CASE state OF
    BAG_DELIVERY_STATES.Idle :                     
													IF _mode = DEVICE_MODES.Manual THEN 
														state := BAG_DELIVERY_STATES.Manual;
													ELSIF NOT iBagNotPresent OR Globals.enableDryCycle THEN
														state := BAG_DELIVERY_STATES.Ready;
													ELSIF iBagNotPresent AND (_amFeedToEye OR _amReverseBag) THEN
														state := BAG_DELIVERY_STATES.FeedToEye;
														_amFeedToEye := FALSE;
													END_IF
													IF jogForwardONS.OSR THEN
														bagFeedMasterMotor.MoveDistance(distance := 30, 
                                                                                    acceleration := accelSetpoint, 
                                                                                    deceleration := decelSetpoint, 
                                                                                    velocity := REAL_TO_INT((1 * Globals.VELOCITY_IPS_MULTIPLIER_20_DEGREE_BAG_DELIVERY)));
														bagFeedRearMotor.MoveDistance(distance := 30, 
                                                                                    acceleration := accelSetpoint, 
                                                                                    deceleration := decelSetpoint, 
                                                                                    velocity := REAL_TO_INT((1 * Globals.VELOCITY_IPS_MULTIPLIER_20_DEGREE_BAG_DELIVERY)));
													ELSIF jogReverseONS.OSR THEN
														bagFeedMasterMotor.MoveDistance(distance := -30, 
                                                                                    acceleration := accelSetpoint, 
                                                                                    deceleration := decelSetpoint, 
                                                                                    velocity := REAL_TO_INT((1 * Globals.VELOCITY_IPS_MULTIPLIER_20_DEGREE_BAG_DELIVERY)));
														bagFeedRearMotor.MoveDistance(distance := -30, 
                                                                                    acceleration := accelSetpoint, 
                                                                                    deceleration := decelSetpoint, 
                                                                                    velocity := REAL_TO_INT((1 * Globals.VELOCITY_IPS_MULTIPLIER_20_DEGREE_BAG_DELIVERY)));
													ELSIF jogForwardONS.OSF OR jogReverseONS.OSF THEN
														bagFeedMasterMotor.Stop();
														bagFeedRearMotor.Stop();
													END_IF
    
	BAG_DELIVERY_STATES.FeedToEye :					//Feed to photoeye if not present
													bagFeedMasterMotor.MoveDistance(distance := feedToPhotoeyeSetpoint, 
                                                                                    acceleration := accelSetpoint, 
                                                                                    deceleration := decelSetpoint, 
                                                                                    velocity := REAL_TO_INT((feedToPhotoeyeSetpoint * Globals.VELOCITY_IPS_MULTIPLIER_20_DEGREE_BAG_DELIVERY)));
													bagFeedRearMotor.MoveDistance(distance := feedToPhotoeyeSetpoint, 
                                                                                    acceleration := accelSetpoint, 
                                                                                    deceleration := decelSetpoint, 
                                                                                    velocity := REAL_TO_INT((feedToPhotoeyeSetpoint * Globals.VELOCITY_IPS_MULTIPLIER_20_DEGREE_BAG_DELIVERY)));
													state := BAG_DELIVERY_STATES.FeedingToEye;
													
	BAG_DELIVERY_STATES.FeedingToEye :				// Stop once photoeye seen
													delay.PT := T#3S;
													delay.IN := TRUE;
													IF NOT iBagNotPresent THEN
														bagFeedMasterMotor.Stop();
														bagFeedRearMotor.Stop();
														state := BAG_DELIVERY_STATES.Idle;
														delay.IN := FALSE;
													END_IF
													IF delay.Q THEN
														state := BAG_DELIVERY_STATES.Fault;
														noBagOverEye.Trigger();
														delay.IN := FALSE;
													END_IF
	
    BAG_DELIVERY_STATES.Reverse :                    // Reverse to break perf
                                                    bagFeedMasterMotor.MoveDistance(distance := reverseDistanceSetpoint, 
                                                                                    acceleration := TO_INT((ABS(reverseDistanceSetpoint) * Globals.STEPS_PER_INCH_20_DEGREE_BAG_DELIVERY) *  accelPercent),
                                                                                    deceleration := TO_INT((ABS(reverseDistanceSetpoint) * Globals.STEPS_PER_INCH_20_DEGREE_BAG_DELIVERY) *  decelPercent), 
                                                                                    velocity := REAL_TO_INT((reverseVelocitySetpoint * Globals.VELOCITY_IPS_MULTIPLIER_20_DEGREE_BAG_DELIVERY)));  
													bagFeedRearMotor.MoveDistance(distance := reverseDistanceSetpoint, 
                                                                                    acceleration := TO_INT((ABS(reverseDistanceSetpoint) * Globals.STEPS_PER_INCH_20_DEGREE_BAG_DELIVERY) *  accelPercent),
                                                                                    deceleration := TO_INT((ABS(reverseDistanceSetpoint) * Globals.STEPS_PER_INCH_20_DEGREE_BAG_DELIVERY) *  decelPercent), 
                                                                                    velocity := REAL_TO_INT((reverseVelocitySetpoint * Globals.VELOCITY_IPS_MULTIPLIER_20_DEGREE_BAG_DELIVERY)));    
                                                        state := BAG_DELIVERY_STATES.Reversing;
                                                    
                                                    
    BAG_DELIVERY_STATES.Reversing :                    // Back up until we see the trailing edge of the bag
														 IF iBagNotPresent OR Globals.enableDryCycle THEN
															delay.PT := T#10MS;
															delay.IN := TRUE;
															IF delay.Q THEN
																bagFeedMasterMotor.Stop();
																bagFeedRearMotor.Stop();
																delay.IN := FALSE;
																delayForReverseFault.IN := FALSE;
																state := BAG_DELIVERY_STATES.ReverseToPrinthead;
															END_IF
														ELSIF bagFeedMasterMotor.CommandAcknowledged AND NOT iBagNotPresent THEN
															delayForReverseFault.PT := T#3000MS;
															delayForReverseFault.IN := TRUE;
															IF delayForReverseFault.Q THEN
																reverseFault.Trigger();
																bagFeedMasterMotor.Stop();
																bagFeedRearMotor.Stop();
															delayForReverseFault.IN := FALSE;
															state := BAG_DELIVERY_STATES.Fault; 
															END_IF
															
														END_IF
											
                                                  
													
	BAG_DELIVERY_STATES.ReverseToPrinthead :                    // Reverse to print head
                                                    bagFeedMasterMotor.MoveDistance(distance := reverseToPrintHeadSetpoint, 
                                                                                    acceleration := TO_INT((ABS(reverseToPrintHeadSetpoint) * Globals.STEPS_PER_INCH_20_DEGREE_BAG_DELIVERY) *  accelPercent),
                                                                                    deceleration := TO_INT((ABS(reverseToPrintHeadSetpoint) * Globals.STEPS_PER_INCH_20_DEGREE_BAG_DELIVERY) *  decelPercent), 
                                                                                    velocity := REAL_TO_INT((reverseVelocitySetpoint * Globals.VELOCITY_IPS_MULTIPLIER_20_DEGREE_BAG_DELIVERY))); 
													bagFeedRearMotor.MoveDistance(distance := reverseToPrintHeadSetpoint, 
                                                                                    acceleration := TO_INT((ABS(reverseToPrintHeadSetpoint) * Globals.STEPS_PER_INCH_20_DEGREE_BAG_DELIVERY) *  accelPercent),
                                                                                    deceleration := TO_INT((ABS(reverseToPrintHeadSetpoint) * Globals.STEPS_PER_INCH_20_DEGREE_BAG_DELIVERY) *  decelPercent), 
                                                                                    velocity := REAL_TO_INT((reverseVelocitySetpoint * Globals.VELOCITY_IPS_MULTIPLIER_20_DEGREE_BAG_DELIVERY)));    
                                                    state := BAG_DELIVERY_STATES.ReversingToPrintHead;
													
	BAG_DELIVERY_STATES.ReversingToPrintHead :                    // Reverse to break perf
                                                   	delay.PT := T#50MS;
													delay.IN := TRUE;
													
													IF delay.Q THEN
														IF bagFeedMasterMotor.CommandAcknowledged AND bagFeedMasterMotor.InPosition THEN
                                                        	state := BAG_DELIVERY_STATES.ReverseDone;
                                                    	END_IF
														delay.IN := FALSE;
													END_IF
                                                    
    BAG_DELIVERY_STATES.ReverseDone :                // We don't print in semi auto or manual mode.  In auto mode if the printer is selected then we move to those states
                                                    IF _mode = DEVICE_MODES.SemiAuto OR _mode = DEVICE_MODES.Manual OR (_mode  = DEVICE_MODES.Auto AND autoFeedDelay.Q) THEN
                                                        IF bagFeedMasterMotor.CommandAcknowledged THEN
															state := BAG_DELIVERY_STATES.FeedBagOut;
                                                        	remainingLength := bagLengthSetpoint;
                                                        	_amFeedBagOut := FALSE;
														END_IF
														
                                                    ELSIF (_mode  = DEVICE_MODES.Auto AND _amWaitForPrinter) THEN
                                                        IF bagFeedMasterMotor.CommandAcknowledged THEN
															state := BAG_DELIVERY_STATES.WaitingForPrinter;
															remainingLength := bagLengthSetpoint - (printLengthSetpoint + printOffsetSetpoint + printerExtraFeedLength);
															_amWaitForPrinter := FALSE;  
														END_IF  
                                                    END_IF
                                                        
                                                    
    BAG_DELIVERY_STATES.WaitingForPrinter :            // 
                                                    IF (_mode  = DEVICE_MODES.Auto AND _amPrinterReady) THEN
														IF printOffsetSetpoint <> 0 THEN
															state := BAG_DELIVERY_STATES.FeedToPrintOffset;
														ELSE
															state := BAG_DELIVERY_STATES.FedToPrintOffset;
														END_IF
                                                        
                                                        _amPrinterReady := FALSE;
                                                    END_IF
                                                        
    BAG_DELIVERY_STATES.FeedToPrintOffset :            // 
                                                    bagFeedMasterMotor.MoveDistance(distance := printOffsetSetpoint, 
                                                                                    acceleration := accelSetpoint, 
                                                                                    deceleration := decelSetpoint, 
                                                                                    velocity := REAL_TO_INT((feedVelocitySetpoint * Globals.VELOCITY_IPS_MULTIPLIER_20_DEGREE_BAG_DELIVERY)));  
													bagFeedRearMotor.MoveDistance(distance := printOffsetSetpoint, 
                                                                                    acceleration := accelSetpoint, 
                                                                                    deceleration := decelSetpoint, 
                                                                                    velocity := REAL_TO_INT((feedVelocitySetpoint * Globals.VELOCITY_IPS_MULTIPLIER_20_DEGREE_BAG_DELIVERY)));  
                                                        state := BAG_DELIVERY_STATES.FeedingToPrintOffset;
                                                    
    BAG_DELIVERY_STATES.FeedingToPrintOffset :        // 
													delay.PT := T#50MS;
													delay.IN := TRUE;
													
													IF delay.Q THEN
														IF bagFeedMasterMotor.CommandAcknowledged AND bagFeedMasterMotor.InPosition THEN
                                                        	state := BAG_DELIVERY_STATES.FedToPrintOffset;
                                                    	END_IF
														delay.IN := FALSE;
													END_IF
                                                    
                                                    
    BAG_DELIVERY_STATES.FedToPrintOffset :            // 
                                                    IF (_mode  = DEVICE_MODES.Auto AND _amStartPrint) THEN
                                                        state := BAG_DELIVERY_STATES.FeedAtPrintSpeed;
                                                        _amStartPrint := FALSE;
                                                    END_IF
                                                    
    BAG_DELIVERY_STATES.FeedAtPrintSpeed :            // 
													delay.PT := delayForPrintFeed;
                                                    delay.IN := TRUE;
													
													IF delay.Q THEN
														bagFeedMasterMotor.MoveDistance(distance := printLengthSetpoint + printerExtraFeedLength, 
                                                                                    acceleration := accelSetpoint, 
                                                                                    deceleration := decelSetpoint, 
                                                                                    velocity := REAL_TO_INT((printVelocitySetpoint * Globals.VELOCITY_IPS_MULTIPLIER_20_DEGREE_BAG_DELIVERY)));  
														bagFeedRearMotor.MoveDistance(distance := printLengthSetpoint + printerExtraFeedLength, 
                                                                                    acceleration := accelSetpoint, 
                                                                                    deceleration := decelSetpoint, 
                                                                                    velocity := REAL_TO_INT((printVelocitySetpoint * Globals.VELOCITY_IPS_MULTIPLIER_20_DEGREE_BAG_DELIVERY)));  
                                                        state := BAG_DELIVERY_STATES.FeedingAtPrintSpeed;
														delay.IN := FALSE;
													END_IF
                                                    
    BAG_DELIVERY_STATES.FeedingAtPrintSpeed :        // 
													delay.PT := T#50MS;
													delay.IN := TRUE;
													IF delay.Q THEN
														IF bagFeedMasterMotor.CommandAcknowledged AND bagFeedMasterMotor.InPosition THEN
                                                        	state := BAG_DELIVERY_STATES.FedAtPrintSpeed;
                                                    	END_IF
														delay.IN := FALSE;
													END_IF
                                                   
                                                    
    BAG_DELIVERY_STATES.FedAtPrintSpeed :            // 
                                                    IF (_mode  = DEVICE_MODES.Auto AND _amPrinterDone) THEN
                                                        state := BAG_DELIVERY_STATES.FeedBagOut;
                                                        _amPrinterDone := FALSE;
                                                    END_IF
                                                    
    BAG_DELIVERY_STATES.FeedBagOut :                // Feed bag length out
                                                    //bagFeedMasterMotor.MoveDistanceFinal(distance := (remainingLength + sealOffsetSetpoint + (reverseToPrintHeadSetpoint*-1)), 
													bagFeedMasterMotor.MoveDistanceFinal(distance := (remainingLength + sealBarToPrintHeadLength) - sealOffsetSetpoint, 
                                                                                        acceleration := accelSetpoint, 
                                                                                        deceleration := decelSetpoint, 
                                                                                        velocity := REAL_TO_INT((feedVelocitySetpoint * Globals.VELOCITY_IPS_MULTIPLIER_20_DEGREE_BAG_DELIVERY)));
													bagFeedRearMotor.MoveDistance(distance := (remainingLength + sealBarToPrintHeadLength) - sealOffsetSetpoint, 
                                                                                        acceleration := accelSetpoint, 
                                                                                        deceleration := decelSetpoint, 
                                                                                        velocity := REAL_TO_INT((feedVelocitySetpoint * Globals.VELOCITY_IPS_MULTIPLIER_20_DEGREE_BAG_DELIVERY)));
                                                    state := BAG_DELIVERY_STATES.FeedingBagOut;    
    
    BAG_DELIVERY_STATES.FeedingBagOut :                // Wait until move is done
													delay.PT := T#50MS;
													delay.IN := TRUE;
													IF delay.Q THEN
														IF bagFeedMasterMotor.CommandAcknowledged AND bagFeedMasterMotor.InPosition THEN
                                                        state := BAG_DELIVERY_STATES.FedBagOut;
														
                                                    	END_IF
														delay.IN := FALSE;
													END_IF
                                                    
    
    BAG_DELIVERY_STATES.FedBagOut :                    // Go to the next ready state
                                                    IF _mode = DEVICE_MODES.Manual THEN 
                                                        state := BAG_DELIVERY_STATES.Manual;
                                                    ELSE
                                                        state := BAG_DELIVERY_STATES.Ready;
                                                    END_IF
													HMIData.driveRollerClean.SetCount(HMIData.driveRollerClean.count + TO_INT(bagLengthSetpoint));
                                                    Globals.bagDeliveryCycleCount := Globals.bagDeliveryCycleCount + 1;
    
    BAG_DELIVERY_STATES.Ready :                        IF (_mode = DEVICE_MODES.Auto AND _amReverseBag) OR _mode = DEVICE_MODES.SemiAuto THEN 
                                                        state := BAG_DELIVERY_STATES.Reverse;
                                                        ClearCommands();
                                                    END_IF 
													_amFeedToEye := FALSE;
													IF iBagNotPresent AND NOT Globals.enableDryCycle THEN 
														state := BAG_DELIVERY_STATES.Idle;
													END_IF
													IF jogForwardONS.OSR THEN
														bagFeedMasterMotor.MoveDistance(distance := 30, 
                                                                                    acceleration := accelSetpoint, 
                                                                                    deceleration := decelSetpoint, 
                                                                                    velocity := REAL_TO_INT((1 * Globals.VELOCITY_IPS_MULTIPLIER_20_DEGREE_BAG_DELIVERY)));
														bagFeedRearMotor.MoveDistance(distance := 30, 
                                                                                    acceleration := accelSetpoint, 
                                                                                    deceleration := decelSetpoint, 
                                                                                    velocity := REAL_TO_INT((1 * Globals.VELOCITY_IPS_MULTIPLIER_20_DEGREE_BAG_DELIVERY)));
													ELSIF jogReverseONS.OSR THEN
														bagFeedMasterMotor.MoveDistance(distance := -30, 
                                                                                    acceleration := accelSetpoint, 
                                                                                    deceleration := decelSetpoint, 
                                                                                    velocity := REAL_TO_INT((1 * Globals.VELOCITY_IPS_MULTIPLIER_20_DEGREE_BAG_DELIVERY)));
														bagFeedRearMotor.MoveDistance(distance := -30, 
                                                                                    acceleration := accelSetpoint, 
                                                                                    deceleration := decelSetpoint, 
                                                                                    velocity := REAL_TO_INT((1 * Globals.VELOCITY_IPS_MULTIPLIER_20_DEGREE_BAG_DELIVERY)));
													ELSIF jogForwardONS.OSF OR jogReverseONS.OSF THEN
														bagFeedMasterMotor.Stop();
														bagFeedRearMotor.Stop();
													END_IF
    
    BAG_DELIVERY_STATES.Fault :                        ClearCommands();
													IF jogForwardONS.OSR THEN
														bagFeedMasterMotor.MoveDistance(distance := 30, 
                                                                                    acceleration := accelSetpoint, 
                                                                                    deceleration := decelSetpoint, 
                                                                                    velocity := REAL_TO_INT((1 * Globals.VELOCITY_IPS_MULTIPLIER_20_DEGREE_BAG_DELIVERY)));
													ELSIF jogReverseONS.OSR THEN
														bagFeedMasterMotor.MoveDistance(distance := -30, 
                                                                                    acceleration := accelSetpoint, 
                                                                                    deceleration := decelSetpoint, 
                                                                                    velocity := REAL_TO_INT((1 * Globals.VELOCITY_IPS_MULTIPLIER_20_DEGREE_BAG_DELIVERY)));
													ELSIF jogForwardONS.OSF OR jogReverseONS.OSF THEN
														bagFeedMasterMotor.Stop();
														bagFeedRearMotor.Stop();
													END_IF
    
    BAG_DELIVERY_STATES.Manual :                    IF _mode = DEVICE_MODES.Auto THEN
														state := BAG_DELIVERY_STATES.Ready;	
													END_IF
													// Manually feed bags out
                                                    IF feedBagPB THEN
                                                        state := BAG_DELIVERY_STATES.Reverse;
                                                        feedBagPB := FALSE;
                                                    END_IF
                                                        
END_CASE

PROPERTY Ready : BOOL
GET
Ready := _ready;
END_GET
SET
_ready := Ready;
END_SET
END_PROPERTY

METHOD PRIVATE ClearCommands
VAR_INPUT
END_VAR
_amFeedBagOut := FALSE;
_amReverseBag := FALSE;
_amPrinterDone := FALSE;
_amPrinterReady := FALSE;
_amWaitForPrinter := FALSE;
_amStartPrint := FALSE;
//_amFeedToEye := FALSE;
END_METHOD

PROPERTY Mode : DEVICE_MODES
SET
_mode := Mode;
END_SET
GET
Mode := _mode;
END_GET
END_PROPERTY

METHOD AutoReverseBag
VAR_INPUT
END_VAR
_amReverseBag := TRUE;
END_METHOD

METHOD AutoPrinterDone
VAR_INPUT
END_VAR
_amPrinterDone := TRUE;
END_METHOD

METHOD AutoWaitForPrinter
VAR_INPUT
END_VAR
_amWaitForPrinter := TRUE;
END_METHOD

METHOD AutoStartPrintFeed
VAR_INPUT
END_VAR
_amStartPrint := TRUE;
END_METHOD

METHOD AutoFeedBagOut
VAR_INPUT
END_VAR
_amFeedBagOut := TRUE;
END_METHOD

METHOD AutoFeedToEye
VAR_INPUT
END_VAR
_amFeedToEye := TRUE;
END_METHOD

METHOD AutoPrinterReady
VAR_INPUT
END_VAR
_amPrinterReady := TRUE;
END_METHOD

END_FUNCTION_BLOCK

// Device/Application/ObjectHandling/IResettable
INTERFACE IResettable EXTENDS IAllObjects

END_INTERFACE

// Device/Application/ObjectHandling/FB_CollectionHandlerLogs
FUNCTION_BLOCK FB_CollectionHandlerLogs
VAR_INPUT
END_VAR
VAR
	Collection: ARRAY[0..GlobalObjects.MAX_LOGS] OF IMachineLogger; // object array
	ObjNames   : ARRAY[0..GlobalObjects.MAX_LOGS] OF STRING;
	_ArrayOver   : BOOL;
	_BadObj      : INT;
	_DupeObj   : INT;
	_OverObj   : INT;
	_TotalObj   : UINT;
END_VAR

METHOD AddObject
VAR_INPUT
	Obj   : IMachineLogger;
END_VAR
VAR
	J   : UINT;
END_VAR
FOR J:= 0 TO _TotalObj DO
	IF Collection[J] = Obj THEN
		// object pointer matches - dupe!
		_DupeObj:= _DupeObj + 1;
		RETURN;
	END_IF
END_FOR
   
IF _TotalObj < GlobalObjects.MAX_LOGS THEN
	Collection[_TotalObj]:= Obj;
	ObjNames[_TotalObj]:= Obj.InstanceName;
	_TotalObj:= _TotalObj + 1;
ELSE
	_ArrayOver:= TRUE;
	_OverObj:= _OverObj + 1;
END_IF
END_METHOD

END_FUNCTION_BLOCK

// Device/Application/ObjectHandling/FB_CollectionHandlerLoggable
FUNCTION_BLOCK FB_CollectionHandlerLoggable
VAR_INPUT

END_VAR
VAR
	Collection: ARRAY[0..GlobalObjects.MAX_LOGGABLE] OF ILoggable; // object array
	ObjNames   : ARRAY[0..GlobalObjects.MAX_LOGGABLE] OF STRING;
	_ArrayOver   : BOOL;
	_BadObj      : INT;
	_DupeObj   : INT;
	_OverObj   : INT;
	_TotalObj   : UINT;
	_internalLogger : REFERENCE TO IMachineLogger;
END_VAR

//	Function Block: FB_CollectionHandlerLoggable
//	Description: This collection handler takes in loggable objects and registers them with a logger.  The FirstScan function should trigger the 
//				 RegisterAll() method to register all loggable objects with a logger
//	Created by: Ben Hess
//	Created Date: Tuesday, September 11, 2018

METHOD RegisterAll
VAR_INPUT
	internalLogger : IMachineLogger;
END_VAR
VAR
	I   : UINT;
	J : UINT;
	cast : ILoggable;
END_VAR
FOR J:= 0 TO _TotalObj - 1 DO
	IF (__QUERYINTERFACE(Collection[J], Cast)) THEN
		cast.RegisterLogger(internalLogger := internalLogger);
	ELSE
		RETURN;
	END_IF
END_FOR
END_METHOD

METHOD AddObject
VAR_INPUT
	Obj   : ILoggable;
END_VAR
VAR
	J   : UINT;
END_VAR
FOR J:= 0 TO _TotalObj DO
	IF Collection[J] = Obj THEN
		// object pointer matches - dupe!
		_DupeObj:= _DupeObj + 1;
		RETURN;
	END_IF
END_FOR
   
IF _TotalObj < GlobalObjects.MAX_LOGGABLE THEN
	Collection[_TotalObj]:= Obj;
	ObjNames[_TotalObj]:= Obj.InstanceName;
	_TotalObj:= _TotalObj + 1;
ELSE
	_ArrayOver:= TRUE;
	_OverObj:= _OverObj + 1;
END_IF
END_METHOD

END_FUNCTION_BLOCK

// Device/Application/Event Handlers/OnlineChangeDone
FUNCTION OnlineChangeDone : DWORD
VAR_IN_OUT
	EventPrm: CmpApp.EVTPARAM_CmpApp;
END_VAR
VAR
END_VAR

RecallValues();

END_FUNCTION

// Project Information/GetCompany
// This function has been automatically generated from the project information.
{attribute 'signature_flag' := '1073741824'}
{attribute 'register_in_runtime'}
FUNCTION GetCompany : WSTRING
VAR_INPUT
	
END_VAR

GetCompany := "Sharp Packaging";

END_FUNCTION

// Library Information/IsLibReleased
// This function has been automatically generated from the project information.
FUNCTION IsLibReleased : BOOL
VAR_INPUT
	
END_VAR

IsLibReleased := FALSE;

END_FUNCTION

// Device/Application/Interfaces/IFaultHandler
INTERFACE IFaultHandler

METHOD AddActiveFault
VAR_INPUT
END_VAR
END_METHOD

METHOD RemoveActiveFault
VAR_INPUT
END_VAR
END_METHOD

END_INTERFACE

// Project Information/GetTitle
// This function has been automatically generated from the project information.
{attribute 'signature_flag' := '1073741824'}
{attribute 'register_in_runtime'}
FUNCTION GetTitle : WSTRING
VAR_INPUT
	
END_VAR

GetTitle := "MOAB Prototype";

END_FUNCTION

// Device/Application/FBs/Motors/Applied Motion/Modbus Commands/FB_SendMoveCommandAppliedMotionRTU
FUNCTION_BLOCK FB_SendMoveCommandAppliedMotionRTU
VAR_INPUT
//    distanceHighWord : WORD;
//    distanceLowWord : WORD;        
//    acceleration : INT;        //Acceleration in RPM/sec
//    deceleration : INT;        //Deceleration in RPM/sec
//    velocity : INT;            //Velocity in .25RPM
    opcode : STEP_SERVO_OPCODES;    //Opcode to perform
    
    //Parameters from motor - we need to check these to verify successful send
    distanceHighWordFromMotor : REFERENCE TO WORD;    //DistanceHighWord From Motor
    distanceLowWordFromMotor : REFERENCE TO WORD;        //DistanceLowWord from Motor
    accelerationFromMotor : REFERENCE TO INT;        //Acceleration in RPM/sec from Motor
    decelerationFromMotor : REFERENCE TO INT;        //Deceleration in RPM/sec from Motor
    velocityFromMotor : REFERENCE TO INT;            //Velocity in .25RPM from Motor
    //opcodeFromMotor : REFERENCE TO INT;                //Opcode from motor
END_VAR
VAR_IN_OUT
    parameterSettingsBuffer : ARRAY [0..4] OF WORD;
END_VAR

VAR_OUTPUT
    triggerParameterWrite : BOOL;
    triggerOpcodeWrite : BOOL;
    xDone : BOOL;
END_VAR
VAR
    moveCommandState : MOVE_MODBUS_COMMAND_STATES;
    modbusRequestTCP: IoDrvModbusTCP.ModbusRequest;
    modbusCommandTCP : IoDrvModbusTCP.ModbusCommand;
    sendBuffer : ARRAY [0 .. 4] OF WORD;            //Array of registers to send
    xExecute : BOOL;
    xExecuteONS : R_TRIG();
END_VAR


xExecuteONS(CLK := xExecute);
IF xExecuteONS.Q THEN
    xDone := FALSE;
END_IF    

CASE moveCommandState OF
    MOVE_MODBUS_COMMAND_STATES.Idle :                    //Move on to Send Parameters
                                                        IF xExecute THEN
                                                            moveCommandState := MOVE_MODBUS_COMMAND_STATES.SendParameters;
                                                        END_IF
                                                        xExecute := FALSE;
                                
    MOVE_MODBUS_COMMAND_STATES.SendParameters :            //We have to use triggers instead of taking over the handle to the COM port
                                                        IF CheckIfParSendSuccessful() THEN
                                                            moveCommandState := MOVE_MODBUS_COMMAND_STATES.SendOpcode;
                                                        ELSE    
                                                            triggerParameterWrite := TRUE;
                                                            moveCommandState := MOVE_MODBUS_COMMAND_STATES.WaitAfterParametersSent;                                            
                                                        END_IF
                                                        
    MOVE_MODBUS_COMMAND_STATES.WaitAfterParametersSent :
                                                        //Wait for confimation
                                                        IF CheckIfParSendSuccessful() THEN
                                                            moveCommandState := MOVE_MODBUS_COMMAND_STATES.SendOpcode;                                                    
                                                        END_IF
    MOVE_MODBUS_COMMAND_STATES.SendOpcode :                
                                                        //Send just Opcode now
                                                        triggerOpcodeWrite := TRUE;
                                                        moveCommandState := MOVE_MODBUS_COMMAND_STATES.WaitAfterOpcodeSent;
                                                        
    MOVE_MODBUS_COMMAND_STATES.WaitAfterOpcodeSent :    //
                                                        xDone := TRUE;
                                                        triggerParameterWrite := FALSE;
                                                        triggerOpcodeWrite := FALSE;
                                                        moveCommandState := MOVE_MODBUS_COMMAND_STATES.Idle;    
                                        
    MOVE_MODBUS_COMMAND_STATES.Fault :                    
                                                        //Move on to Send Parameters
                                                        IF xExecute THEN
                                                            moveCommandState := MOVE_MODBUS_COMMAND_STATES.SendParameters;
                                                        END_IF
                                                        xExecute := FALSE;
END_CASE

METHOD Execute
VAR_INPUT
END_VAR
xExecute := TRUE;
END_METHOD

METHOD CheckIfParSendSuccessful : BOOL
VAR_INPUT
END_VAR

//Check to make sure we have a valid reference.  Disable complier warning since we're doing the check
{warning disable C0371}
IF NOT __ISVALIDREF(parameterSettingsBuffer) THEN
     RETURN;
END_IF

//Check if parameters from drive match the ones we sent

CheckIfParSendSuccessful := (parameterSettingsBuffer[0] = INT_TO_WORD(accelerationFromMotor) AND parameterSettingsBuffer[1] = INT_TO_WORD(decelerationFromMotor) AND parameterSettingsBuffer[2] = INT_TO_WORD(velocityFromMotor) AND parameterSettingsBuffer[3] = distanceHighWordFromMotor AND parameterSettingsBuffer[4] = distanceLowWordFromMotor);
{warning restore C0371}
END_METHOD

END_FUNCTION_BLOCK

// Device/Application/FBs/Motors/Applied Motion/FB_AppliedMotionStepServoEIPPassthrough_1
FUNCTION_BLOCK FB_AppliedMotionStepServoEIPPassthrough_1 EXTENDS FB_AppliedMotionStepServoEIPPassthrough
VAR_INPUT
END_VAR
VAR_OUTPUT
END_VAR
VAR
END_VAR

SUPER^();

METHOD DoneClamping
VAR_INPUT
END_VAR
END_METHOD

METHOD AllowClamping
VAR_INPUT
END_VAR
MoveDistanceTorque(velocity:=100, acceleration := 1, deceleration := 1, distance := 0, current := 1);
END_METHOD

END_FUNCTION_BLOCK

// Device/Application/FBs/FB_PredictiveMaint
FUNCTION_BLOCK FB_PredictiveMaint EXTENDS FB_CycleCounter
VAR_INPUT
	target : UDINT;
	name : STRING;
	units : STRING := 'Machine Cycles';
END_VAR
VAR_OUTPUT
	
END_VAR
VAR
	
END_VAR

SUPER^();

END_FUNCTION_BLOCK

// Device/Application/FBs/FB_CycleCounter
FUNCTION_BLOCK FB_CycleCounter
VAR_INPUT
	reset : BOOL;
END_VAR
VAR_OUTPUT
END_VAR
VAR
    count : UDINT;
END_VAR

IF reset THEN
	THIS^.Clear();
	reset := FALSE;
END_IF

METHOD Increment
VAR_INPUT
END_VAR
count := count + 1;
END_METHOD

METHOD Clear
VAR_INPUT
END_VAR
count := 0;
END_METHOD

METHOD SetCount
VAR_INPUT
	countSetting : UDINT;
END_VAR
count := countSetting;
END_METHOD

END_FUNCTION_BLOCK

// Device/Application/FBs/Motors/Applied Motion/FB_AppliedMotionBagDeliveryMotorNoFollowing
FUNCTION_BLOCK FB_AppliedMotionBagDeliveryMotorNoFollowing EXTENDS FB_AppliedMotionStepServoEIPBase
VAR_INPUT
END_VAR
VAR_OUTPUT
END_VAR
VAR
	_moveDistance : BOOL;
	_moveDistanceONS : R_TRIG;
	_moveFinal : BOOL;
	_moveFinalONS : R_TRIG;
	_moveDone : BOOL;
	waitForMove : TON := (PT := T#30MS);
	manualFinalMovePB : BOOL;
	movedFinal : BOOL;
	moveDistanceState : AMP_EIP_MOVE_INITIAL_STATES;
	moveDistanceFinalState : AMP_EIP_MOVE_INITIAL_STATES;
END_VAR

METHOD MoveDistance
VAR_INPUT
    distance : REAL;        //Distance to move in inches
    acceleration : INT;        //Acceleration in RPM/sec
    deceleration : INT;        //Deceleration in RPM/sec
    velocity : INT;            //Velocity in .25RPM
END_VAR
commandSuccessful := FALSE;
_moveDone := FALSE;
moveDistanceState := AMP_EIP_MOVE_INITIAL_STATES.Idle;
distanceToMoveInSteps := REAL_TO_DINT((distance) * stepsPerInchSetpoint);

IF reversePolarity THEN
    distanceToMoveInSteps := distanceToMoveInSteps * -1;
END_IF

pointToPointAccelSetpoint := acceleration;
pointToPointDecelSetpoint := deceleration;
velocitySetpoint := velocity;

currentLimit := defaultCurrentSetpoint;
_moveDistance := TRUE;

//commands.feedToLength := TRUE;
//SUPER^.ExecuteStoredProgram(1);
END_METHOD

METHOD SetRearMotorToTorqueMode
VAR_INPUT
END_VAR
END_METHOD

METHOD Execute
VAR_INPUT
END_VAR
SUPER^.Execute();
waitForMove();
_moveDistanceONS(CLK := _moveDistance);
_moveFinalONS(CLK := _moveFinal);

CASE moveDistanceState OF
	AMP_EIP_MOVE_INITIAL_STATES.Idle :						
															IF _moveDistance THEN
																moveDistanceState := AMP_EIP_MOVE_INITIAL_STATES.SetOutputOff;
															END_IF
															
	AMP_EIP_MOVE_INITIAL_STATES.SetOutputOff :					sclCommand := 16#534F; //Output off
															parameter1 := 16#48B2;
															commands.SendHostCommand := TRUE;
															IF commandSuccessful THEN
																commandSuccessful := FALSE;
																moveDistanceState := AMP_EIP_MOVE_INITIAL_STATES.WaitAfterSettingOutputOff;
															END_IF
															
	AMP_EIP_MOVE_INITIAL_STATES.WaitAfterSettingOutputOff :		
															IF commandSuccessful THEN
																moveDistanceState := AMP_EIP_MOVE_INITIAL_STATES.MoveMotor;
															END_IF
																
	AMP_EIP_MOVE_INITIAL_STATES.MoveMotor: 					commandSuccessful := FALSE;
															sclCommand := 16#0;
															parameter1 := 16#0;
															commands.FeedToLength := TRUE;
															_moveDistance := FALSE;
															moveDistanceState := AMP_EIP_MOVE_INITIAL_STATES.WaitAfterMovingMotor;
															
															
	AMP_EIP_MOVE_INITIAL_STATES.WaitAfterMovingMotor: 		IF commandSuccessful THEN
																_moveDone := TRUE;
																moveDistanceState := AMP_EIP_MOVE_INITIAL_STATES.Idle;
															END_IF														
END_CASE

CASE moveDistanceFinalState OF
	AMP_EIP_MOVE_INITIAL_STATES.Idle :						IF _moveFinal THEN
																moveDistanceFinalState := AMP_EIP_MOVE_INITIAL_STATES.MoveMotor;
															END_IF
	
	AMP_EIP_MOVE_INITIAL_STATES.MoveMotor: 					sclCommand := 16#0;
															parameter1 := 16#0;
															commandSuccessful := FALSE;	
															commands.FeedToLength := TRUE;
															moveDistanceFinalState := AMP_EIP_MOVE_INITIAL_STATES.WaitAfterMovingMotor;
															
															
	AMP_EIP_MOVE_INITIAL_STATES.WaitAfterMovingMotor: 		IF commandSuccessful AND InPosition THEN	
																moveDistanceFinalState := AMP_EIP_MOVE_INITIAL_STATES.SetOutputOff;
															END_IF
														
	AMP_EIP_MOVE_INITIAL_STATES.SetOutputOff :					sclCommand := 16#534F; // Output on
															parameter1 := 16#4CB2;
															
															commandSuccessful := FALSE;
															commands.SendHostCommand := TRUE;
															_moveFinal := FALSE;
															moveDistanceFinalState := AMP_EIP_MOVE_INITIAL_STATES.WaitAfterSettingOutputOff;
															
															
	AMP_EIP_MOVE_INITIAL_STATES.WaitAfterSettingOutputOff :		
															IF commandSuccessful THEN
																_moveDone := TRUE;
																moveDistanceFinalState := AMP_EIP_MOVE_INITIAL_STATES.Idle;
															END_IF
																

END_CASE
(*
IF _moveFinal THEN	
	IF NOT movedFinal AND commandSuccessful THEN
		commandSuccessful := FALSE;
		commands.FeedToLength := TRUE;
		waitForMove.IN := TRUE;
		movedFinal := TRUE;
	END_IF
	
	IF commandSuccessful AND waitForMove.Q AND InPosition THEN
		sclCommand := 16#534F;
		parameter1 := 16#4CB2;
		commands.SendHostCommand := TRUE;
		_moveFinal := FALSE;
		waitForMove.IN := FALSE;
		movedFinal := FALSE;
	END_IF
END_IF
*)
IF manualFinalMovePB THEN
    MoveDistanceFinal(distance := distanceSetpointInches, acceleration := pointToPointAccelSetpoint, deceleration := pointToPointDecelSetpoint, velocity := velocitySetpoint);
    manualFinalMovePB := FALSE;
END_IF
END_METHOD

METHOD SetRearMotorToEncoderFollowing
VAR_INPUT
END_VAR
END_METHOD

METHOD MoveDistanceFinal
VAR_INPUT
    distance : REAL;        //Distance to move in inches
    acceleration : INT;        //Acceleration in RPM/sec
    deceleration : INT;        //Deceleration in RPM/sec
    velocity : INT;            //Velocity in .25RPM
END_VAR
commandSuccessful := FALSE;
_moveDone := FALSE;
moveDistanceFinalState := AMP_EIP_MOVE_INITIAL_STATES.Idle;
distanceToMoveInSteps := REAL_TO_DINT((distance) * stepsPerInchSetpoint);
IF reversePolarity THEN
    distanceToMoveInSteps := distanceToMoveInSteps * -1;
END_IF

pointToPointAccelSetpoint := acceleration;
pointToPointDecelSetpoint := deceleration;
velocitySetpoint := velocity;

currentLimit := defaultCurrentSetpoint;
_moveFinal := TRUE;
//SUPER^.ExecuteStoredProgram(2);
END_METHOD

PROPERTY CommandAcknowledged : BOOL
GET
CommandAcknowledged := _moveDone;
END_GET
END_PROPERTY

METHOD StopViaProgram
// Load program segment 12 into buffer and execute.  This program contains nothing but a SM command.
// We must do it this way because the normal "stop command" opcode we have access to over modbus 
// also kills the program buffer which is bad.
SUPER^.Stop();
END_METHOD

END_FUNCTION_BLOCK

// Device/Application/ObjectHandling/FB_CollectionHandlerInitializable
FUNCTION_BLOCK FB_CollectionHandlerInitializable
VAR_INPUT

END_VAR
VAR
	Collection: ARRAY[0..GlobalObjects.MAX_LOGGABLE] OF IInitializable; // object array
	ObjNames   : ARRAY[0..GlobalObjects.MAX_LOGGABLE] OF STRING;
	_ArrayOver   : BOOL;
	_BadObj      : INT;
	_DupeObj   : INT;
	_OverObj   : INT;
	_TotalObj   : UINT;
END_VAR

//	Function Block: FB_CollectionHandlerLoggable
//	Description: This collection handler takes in loggable objects and registers them with a logger.  The FirstScan function should trigger the 
//				 RegisterAll() method to register all loggable objects with a logger
//	Created by: Ben Hess
//	Created Date: Tuesday, September 11, 2018

METHOD InitializeAll
VAR_INPUT
	
END_VAR
VAR
	J : UINT;
	Cast : IInitializable;
END_VAR
FOR J:= 0 TO _TotalObj - 1 DO
	IF (__QUERYINTERFACE(Collection[J], Cast)) THEN
		Cast.Initialize();
	ELSE 
		RETURN;
	END_IF
END_FOR
END_METHOD

METHOD AddObject
VAR_INPUT
	Obj   : IInitializable;
END_VAR
VAR
	J   : UINT;
END_VAR
FOR J:= 0 TO _TotalObj DO
	IF Collection[J] = Obj THEN
		// object pointer matches - dupe!
		_DupeObj:= _DupeObj + 1;
		RETURN;
	END_IF
END_FOR
   
IF _TotalObj < GlobalObjects.MAX_LOGGABLE THEN
	Collection[_TotalObj]:= Obj;
	ObjNames[_TotalObj]:= Obj.InstanceName;
	_TotalObj:= _TotalObj + 1;
ELSE
	_ArrayOver:= TRUE;
	_OverObj:= _OverObj + 1;
END_IF
END_METHOD

END_FUNCTION_BLOCK

// Device/Application/Event Handlers/PrepareShutdown
FUNCTION PrepareShutdown : DWORD
VAR_IN_OUT
	EventPrm: Component_Manager.EVTPARAM_CmpMgr_Shutdown;
END_VAR
VAR
END_VAR

SaveValues();

END_FUNCTION

// Device/Application/FBs/Cylinders/FB_ThreePositionCylinderWithFeedback
FUNCTION_BLOCK FB_ThreePositionCylinderWithFeedback EXTENDS FB_Cylinder IMPLEMENTS ICylinder, IThreePositonCylinder, IFault
VAR_INPUT
    extendedFeedbackInput : BOOL;    //Extended feedback input from I/O
    retractedFeedbackInput : BOOL;    //Retracted feedback input from I/O
    extendFaultDelay : INT := 1000;        //Extend fault delay in MS
    retractFaultDelay : INT := 1000;        //Retract fault delay in MS
    faultMonitoring : BOOL;                    //Fault monitoring enabled if true
END_VAR
VAR_OUTPUT
    failedToExtend : BOOL;            //Failed to Extend Fault
    failedToRetract : BOOL;            //Failed to Retract Fault
END_VAR
VAR
    faultIndication : BOOL;            //Overall fault status of cylinder
    extendFaultTimer : TON;            //Extend Fault Timer
    retractFaultTimer : TON;        //Retract Fault Timer
    resetFaults : BOOL;                //Reset faults
END_VAR

METHOD ResetFault
//Reset all faults
failedToExtend := FALSE;
failedToRetract := FALSE;
END_METHOD

METHOD Exhaust
extendOutput := FALSE;
retractOutput := FALSE;
END_METHOD

METHOD Execute
//This code monitors the positon of the cylinder and raises a fault if the cylinder doesn't reach its
//desired postion within the specified time.

//Initialize timers
extendFaultTimer(PT := INT_TO_TIME(extendFaultDelay));
retractFaultTimer(PT := INT_TO_TIME(retractFaultDelay));

//Only enable timers if we are to be monitoring faults
IF faultMonitoring THEN
    extendFaultTimer.IN := (extendOutput AND NOT extendedFeedbackInput);
    retractFaultTimer.IN := (retractOutput AND NOT retractedFeedbackInput);
ELSE 
        extendFaultTimer.IN := FALSE;
        retractFaultTimer.IN := FALSE;
END_IF

//Rasie the alarms
failedToExtend S= extendFaultTimer.Q;
failedToRetract S= retractFaultTimer.Q;

//Set overall fault indication
faultIndication := failedToExtend OR failedToRetract;
END_METHOD

PROPERTY Faulted : BOOL
SET
faultIndication := Faulted;
END_SET
GET
Faulted := faultIndication;
END_GET
END_PROPERTY

END_FUNCTION_BLOCK

// Device/Application/FBs/FB_CylinderLeak
FUNCTION_BLOCK FB_CylinderLeak EXTENDS FB_PredictiveMaint
VAR_INPUT
	iExtended : BOOL;
	iRetracted : BOOL;
	maximumStrokeTime : REAL;
END_VAR
VAR_OUTPUT
	strokeTime : REAL;
END_VAR
VAR
	strokeTimer : TON := (PT := T#1H);
	extendedONS : R_TRIG;
	retractedONS : R_TRIG;
END_VAR

extendedONS(CLK := iExtended);
retractedONS(CLK := iRetracted);

IF extendedONS.Q OR retractedONS.Q THEN
	strokeTime := TO_REAL(strokeTimer.ET) / 1000;
END_IF

strokeTimer(IN := NOT iExtended AND NOT iRetracted);

END_FUNCTION_BLOCK

// Device/Application/FBs/FB_DriveTemp
FUNCTION_BLOCK FB_DriveTemp EXTENDS FB_PredictiveMaint
VAR_INPUT
	iDriveTemp : DINT;
	maxTemp : REAL;
END_VAR
VAR_OUTPUT
	DriveTemp : REAL;
END_VAR
VAR
END_VAR

DriveTemp := TO_REAL(iDriveTemp) / 10.0;

END_FUNCTION_BLOCK

// Device/Application/ObjectHandling/FB_CollectionHandlerActiveFaults
FUNCTION_BLOCK FB_CollectionHandlerActiveFaults
VAR_INPUT
END_VAR
VAR
	Collection: ARRAY[0..GlobalObjects.MAX_FAULTS] OF IFault; // object array
	ObjNames   : ARRAY[0..GlobalObjects.MAX_FAULTS] OF STRING;
	_ArrayOver   : BOOL;
	_BadObj      : INT;
	_DupeObj   : INT;
	_OverObj   : INT;
	_TotalObj   : UINT;
END_VAR

VAR_OUTPUT
	faultActive : BOOL;
END_VAR

//	Function Block: FB_CollectionHandlerActiveFaults
//	Description: This collection handler adds and removes active faults to an array
//				 The add and remove methods are called from FB_Fault
//	Created by: Tom Jacobs
//	Created Date: Friday, September 7, 2018

METHOD RemoveObject
VAR_INPUT
	Obj   : IFault;
END_VAR

VAR
	I   : UINT;
	J : UINT;
END_VAR
FOR I:= 0 TO _TotalObj DO
	IF Collection[I] = Obj THEN
		// object pointer matches - get rid of it
		FOR J := I TO _TotalObj DO
			Collection[J] := Collection[J+1];
			ObjNames[J]:= ObjNames[J+1]; 
		END_FOR
		_TotalObj := _TotalObj - 1;
		IF _TotalObj = 0 THEN
			faultActive := FALSE;
		END_IF
		RETURN;
	END_IF
END_FOR
END_METHOD

METHOD AckAll
VAR_INPUT
END_VAR
VAR
	Cast : IFault;
	Fault : IFault;
	J : UINT;
END_VAR
// For each active fault in the array, ack it.
FOR J:= 0 TO _TotalObj - 1 DO
	IF (__QUERYINTERFACE(Collection[J], Cast)) THEN
		Cast.Ack();
	ELSE 
		RETURN;
	END_IF
END_FOR
END_METHOD

METHOD AddObject
VAR_INPUT
	Obj   : IFault;
END_VAR
VAR
	I   : UINT;
	J : UINT;
END_VAR
// Add the active fault to the array 
FOR J:= 0 TO _TotalObj DO
	IF Collection[J] = Obj THEN
		// object pointer matches - it's already in here
		RETURN;
	END_IF
END_FOR
   
IF _TotalObj < GlobalObjects.MAX_FAULTS THEN
	Collection[_TotalObj]:= Obj;
	ObjNames[_TotalObj]:= Obj.InstanceName;
	_TotalObj:= _TotalObj + 1;
ELSE
	_ArrayOver:= TRUE;
	_OverObj:= _OverObj + 1;
END_IF

faultActive := TRUE;
END_METHOD

END_FUNCTION_BLOCK

// Project Information/GetTextProperty2
// This function has been automatically generated from the project information.
{attribute 'signature_flag' := '1073741824'}
{attribute 'register_in_runtime'}
FUNCTION GetTextProperty2 : POINTER TO WSTRING
VAR_INPUT
	stKey: WSTRING;
END_VAR

IF stKey = "Author" THEN
	GetTextProperty2 := ADR("Ben Hess");
ELSIF stKey = "Company" THEN
	GetTextProperty2 := ADR("Sharp Packaging");
ELSIF stKey = "Project" THEN
	GetTextProperty2 := ADR("AlphaController");
ELSIF stKey = "Title" THEN
	GetTextProperty2 := ADR("MOAB Prototype");
ELSIF stKey = "VersionPostfix" THEN
	GetTextProperty2 := ADR("-alpha/pro24");
ELSE
	GetTextProperty2 := ADR("");
END_IF

END_FUNCTION

// Device/Application/FBs/DataHandlers/FB_ModbusDWORD
FUNCTION_BLOCK FB_ModbusDWORD
VAR_INPUT
END_VAR
VAR_OUTPUT
END_VAR
VAR
    _highWord : WORD;
    _lowWord : WORD;
    _rawValue : DWORD;
END_VAR

//    Function Block: FB_ModbusDWORD
//    Description: Automatically handles the packing and unpacking of Upper and Lower words to create a DWORD
//    for 16 bit modbus communications
//    
//    Created by: Ben Hess
//    Created Date: Wednesday, April 11, 2018

PROPERTY HighWord : WORD
GET
HighWord := _highWord;
END_GET
SET
_highWord := HighWord;
END_SET
END_PROPERTY

PROPERTY RawValue : DWORD
GET
_rawValue := OSCAT_BASIC.DWORD_OF_WORD(_highWord,_lowWord);
RawValue := _rawValue;
END_GET
SET
_rawValue := RawValue;
_highWord := OSCAT_BASIC.WORD_OF_DWORD(in := _rawValue, N := 1);
_lowWord := OSCAT_BASIC.WORD_OF_DWORD(in := _rawValue, N := 0);
END_SET
END_PROPERTY

PROPERTY LowWord : WORD
GET
LowWord := _lowWord;
END_GET
SET
_lowWord := LowWord;
END_SET
END_PROPERTY

END_FUNCTION_BLOCK

// Project Information/GetBooleanProperty
// This function has been automatically generated from the project information.
{attribute 'signature_flag' := '1073741824'}
{attribute 'register_in_runtime'}
FUNCTION GetBooleanProperty : BOOL
VAR_INPUT
	stKey: WSTRING;
END_VAR

GetBooleanProperty := FALSE;

END_FUNCTION

// Device/Application/FBs/Components/PneumaticPressureBarFB
FUNCTION_BLOCK PneumaticPressureBarFB
VAR_INPUT
    enable : BOOL;                    // Enable Pneumatic pressure bar
    sealBarEnable : BOOL;            //Enable seal bar
    bagOpenFingersEnable : BOOL;        //Enable bag open fingers
	iPressureBarRetracted : BOOL;
	iPressureBarExtended : BOOL;
END_VAR
VAR_OUTPUT
    state : PRESSURE_BAR_STATES;     //Jaw State
	oPositionBagOpenFingersToRelease : BOOL;
	oExtendSealBar : BOOL;
	oExtendCylinder : BOOL;
	oRetractCylinder : BOOL;
END_VAR
VAR
    _mode : DEVICE_MODES;            // Auto-SemiAuto-Manual
    _ready : BOOL;                    // Ready to be controlled
    _amOpenJaw : BOOL;    // Auto Mode Open Jaw Command
    _amCloseJaw : BOOL;     // Auto Mode Close Jaw Command
	_amSealBag : BOOL;		// Auto mode seal bag command
    enableONS : R_TRIG; //Enable One Shot
    //autoModeSelect : BOOL;            //Auto Mode Selection (Timers)
    startCyclePB : BOOL;                //Start Cycle
    stopCyclePB : BOOL;                //Stop Cycle
    manualExtendHighPressurePB : BOOL;            //Manually Extend Cylinder High Pressure
    manualExtendLowPressurePB : BOOL;            //Manually Extend Cylinder Low Pressure
    manualRetractPB : BOOL;            //Manually Retract Cylinder
    manualExhaustPB : BOOL;            //Manually Echaust Cylinder
    timerExtendedDebounce : TON;            //Timer for extend delay
    timerExtendDwell : TON;            //Timer for extend dwell after extended
    timerRetractedDebounce : TON;        //Timer for retract delay
    timerRetractDwell : TON;        //Timer for retract dwell after extended
    timerSealDwell : TON;            //Timer for seal dwell
    extendDelaySP : INT := 50;    //Extend delay SP
    extendDwellSP : INT := 300;    //Extend dwell SP
    retractDelaySP : INT := 50;        //Retract delay SP
    retractDwellSP : INT := 750;    //Retract dwell SP
    incrementCount : R_TRIG();
    
    bagOpenFingersReleaseDelay : TON := (PT := T#100MS);                //Delay to open Bag Open Fingers after closing pressure bar
    bagOpenFingersGrabDelay : TON := (PT := T#100MS);                //Delay to close Bag Open Fingers after opening pressure bar
    bagOpenFingers : BagOpenFingersFB();
    openingBag : BOOL;                        //Opening bag flag for bag open fingers  
    incrementSealBarCountONS : Standard.R_TRIG;
    incrementBagOpenFinersONS : Standard.R_TRIG;
    autoModeSelected : BOOL;
    semiAutoModeSelected : BOOL;
    manualModeSelected : BOOL;
END_VAR
VAR_IN_OUT
	
END_VAR

//    Function Block: Cylinder
//    Description: This program moves a jaw cylinder back and forth
//    Created by: Ben Hess
//    Created Date: January 16th, 2017

bagOpenFingers(releaseOutput => oPositionBagOpenFingersToRelease);


//Stop the auto cycle if button pressed or coming out of auto mode or moving the servo.
IF stopCyclePB OR NOT (_mode = DEVICE_MODES.SemiAuto) THEN 
    startCyclePB := FALSE;
END_IF

autoModeSelected := (_mode = DEVICE_MODES.Auto);
semiAutoModeSelected := (_mode = DEVICE_MODES.SemiAuto);
manualModeSelected := (_mode = DEVICE_MODES.Manual);

timerExtendedDebounce(PT := INT_TO_TIME(extendDelaySP));
timerExtendDwell(PT := INT_TO_TIME(extendDwellSP));
timerRetractedDebounce(PT := INT_TO_TIME(retractDelaySP));
timerRetractDwell(PT := INT_TO_TIME(retractDwellSP));
bagOpenFingersReleaseDelay();    
bagOpenFingersGrabDelay();

//Go to idle when enabled
enableONS(CLK := enable);
IF enableONS.Q THEN    
    state := PRESSURE_BAR_STATES.Idle;
END_IF

IF NOT enable THEN
    state := PRESSURE_BAR_STATES.Idle;
END_IF

_ready := (_mode = DEVICE_MODES.Auto) AND NOT (state = PRESSURE_BAR_STATES.Fault);


CASE state OF
    
                                    
    PRESSURE_BAR_STATES.Idle :                //Initial state
                                    IF (semiAutoModeSelected AND startCyclePB) OR (autoModeSelected AND _amOpenJaw) THEN
                                        state := PRESSURE_BAR_STATES.OpenJaw;
                                        _amOpenJaw := FALSE;
                                    ELSIF (autoModeSelected AND _amCloseJaw) THEN
                                        state := PRESSURE_BAR_STATES.CloseJaw;
										_amCloseJaw := FALSE;
                                    ELSIF manualModeSelected THEN
                                        state := PRESSURE_BAR_STATES.Manual;
                                    END_IF
                                    oExtendSealBar := FALSE;
                                    
    
    PRESSURE_BAR_STATES.OpenJaw :                //Open jaw by extending cylinder
                                    ExtendCylinderHighPressure();
                                    state := PRESSURE_BAR_STATES.OpeningJaw;
    
    PRESSURE_BAR_STATES.OpeningJaw :            //
                                    //This delay is a debounce for the sensors.
                                    IF iPressureBarExtended THEN
                                        timerExtendedDebounce.IN := TRUE;
                                        IF timerExtendedDebounce.Q THEN
                                            state := PRESSURE_BAR_STATES.JawOpened;
                                            timerExtendedDebounce.IN := FALSE;
                                        END_IF
                                    END_IF
                                    //If we are opening bag this cycle then grab it now
                                    bagOpenFingersGrabDelay.IN := bagOpenFingersEnable;
                                    IF bagOpenFingersGrabDelay.Q THEN
                                        bagOpenFingers.Grab();
                                        bagOpenFingersGrabDelay.IN := FALSE;
                                    END_IF
                                    
                                    
    
    PRESSURE_BAR_STATES.JawOpened :            //Jaw is opened.  If in semi auto mode, go to close jaw after extend dwell. 
                                    IF (semiAutoModeSelected AND startCyclePB) OR (autoModeSelected AND _amCloseJaw) THEN
                                        timerExtendDwell.IN := TRUE;
                                    END_IF
                                    
                                    IF timerExtendDwell.Q  THEN
                                        state := PRESSURE_BAR_STATES.CloseJaw;
                                        _amCloseJaw := FALSE;
                                        timerExtendDwell.IN := FALSE;
                                    END_IF
    
    PRESSURE_BAR_STATES.CloseJaw :            //Close jaw by retracting cylinder
                                    RetractCylinder();
                                    state := PRESSURE_BAR_STATES.ClosingJaw;
    
    PRESSURE_BAR_STATES.ClosingJaw :            //
                                    //This delay is a debounce after the sensor is seen
                                    IF iPressureBarRetracted THEN
                                        timerRetractedDebounce.IN := TRUE;    
                                        IF timerRetractedDebounce.Q THEN
                                            state := PRESSURE_BAR_STATES.JawClosed;
                                            timerRetractedDebounce.IN := FALSE;
                                        END_IF
                                    END_IF
                                    
                                    
                                    
    
    PRESSURE_BAR_STATES.JawClosed :            //Go to sealing if seal bar enabled, otherwise if in auto mode go to open jaw after retract dwell. Else go back to idle
                                    IF sealBarEnable THEN
                                        state := PRESSURE_BAR_STATES.Sealing;
                                    END_IF
                                    
                                    IF (semiAutoModeSelected AND startCyclePB) OR (autoModeSelected AND _amOpenJaw) THEN
                                        bagOpenFingersReleaseDelay.IN := bagOpenFingersEnable;
                                        timerRetractDwell.IN := TRUE;
                                    END_IF    
                                    
                                    IF bagOpenFingersReleaseDelay.Q THEN
                                        bagOpenFingers.Release();
                                        bagOpenFingersReleaseDelay.IN := FALSE;
                                    END_IF    
                                    
                                    IF timerRetractDwell.Q THEN
                                        state := PRESSURE_BAR_STATES.OpenJaw;
                                        _amOpenJaw := FALSE;
                                        timerRetractDwell.IN := FALSE;
                                    END_IF

    PRESSURE_BAR_STATES.Sealing :                //Seal sets output for seal bar after closed for a dwell setpoint  Hack for now
                                    timerRetractDwell.IN := TRUE;
                                    
                                    IF (semiAutoModeSelected OR (autoModeSelected AND _amOpenJaw)) AND timerRetractDwell.Q THEN
                                        state := PRESSURE_BAR_STATES.OpenJaw;
                                        timerRetractDwell.IN := FALSE;
                                        _amOpenJaw := FALSE;
                                    END_IF
                                    
                                    bagOpenFingersReleaseDelay.IN := bagOpenFingersEnable;
                                    IF bagOpenFingersReleaseDelay.Q THEN
                                        bagOpenFingers.Release();
                                        bagOpenFingersReleaseDelay.IN := FALSE;
                                    END_IF    
                                        
                                    oExtendSealBar := TIME_TO_REAL(timerRetractDwell.ET) > (retractDwellSP * 0.1) AND TIME_TO_REAL(timerRetractDwell.ET) < (retractDwellSP * 0.8);
    
    PRESSURE_BAR_STATES.Manual :    IF manualExhaustPB THEN
                                        ExhaustCylinder();
                                        manualExhaustPB := FALSE;
                                    ELSIF manualRetractPB THEN
                                        RetractCylinder();
                                        manualRetractPB := FALSE;
                                    ELSIF manualExtendHighPressurePB THEN
                                        ExtendCylinderHighPressure();
                                        manualExtendHighPressurePB := FALSE;
									ELSIF manualExtendLowPressurePB THEN
                                        ExtendCylinderLowPressure();
                                        manualExtendLowPressurePB := FALSE;
                                    END_IF
                                
    PRESSURE_BAR_STATES.Fault : 
    
END_CASE

//Count cycles
incrementCount(CLK :=timerExtendDwell.Q); 
IF incrementCount.Q THEN
    Globals.headCycleCount := Globals.headCycleCount + 1;
END_IF

incrementSealBarCountONS(CLK := oExtendSealBar);
IF incrementSealBarCountONS.Q THEN
    Globals.sealBarCount := Globals.sealBarCount + 1;
END_IF

incrementBagOpenFinersONS(CLK := oPositionBagOpenFingersToRelease);
IF incrementBagOpenFinersONS.Q THEN
    Globals.bagOpenFingersCount := Globals.bagOpenFingersCount + 1;
END_IF

METHOD AutoDoneMovingPassthrough
VAR_INPUT
END_VAR
state := PRESSURE_BAR_STATES.Idle;
END_METHOD

METHOD AutoMovingPassthrough
VAR_INPUT
END_VAR
state := PRESSURE_BAR_STATES.Manual;
END_METHOD

METHOD ExhaustCylinder
VAR_INPUT
END_VAR
oExtendCylinder := FALSE;
oRetractCylinder := FALSE;
END_METHOD

PROPERTY Ready : BOOL
GET
Ready := _ready;
END_GET
SET
_ready := Ready;
END_SET
END_PROPERTY

PROPERTY Mode : DEVICE_MODES
SET
_mode := Mode;
END_SET
GET
Mode := _mode;
END_GET
END_PROPERTY

METHOD AutoCloseJaw
VAR_INPUT
END_VAR
_amCloseJaw := TRUE;
END_METHOD

METHOD ExtendCylinderHighPressure
VAR_INPUT
END_VAR
oExtendCylinder := TRUE;
oRetractCylinder := FALSE;
END_METHOD

METHOD ExtendCylinderLowPressure
VAR_INPUT
END_VAR
oExtendCylinder := TRUE;
oRetractCylinder := TRUE;
END_METHOD

METHOD AutoOpenJaw
VAR_INPUT
END_VAR
_amOpenJaw := TRUE;
END_METHOD

METHOD RetractCylinder
VAR_INPUT
END_VAR
oExtendCylinder := FALSE;
oRetractCylinder := TRUE;
END_METHOD

METHOD AutoSealBag
VAR_INPUT
END_VAR
END_METHOD

END_FUNCTION_BLOCK

// Project Information/GetVersionProperty
// This function has been automatically generated from the project information.
{attribute 'signature_flag' := '1073741824'}
{attribute 'register_in_runtime'}
FUNCTION GetVersionProperty : VERSION
VAR_INPUT
	stKey: WSTRING;
END_VAR

IF stKey = "Version" THEN
	GetVersionProperty.uiMajor := 0;
	GetVersionProperty.uiMinor := 9;
	GetVersionProperty.uiServicePack := 13;
	GetVersionProperty.uiPatch := 2;
ELSE
	GetVersionProperty.uiMajor := 0;
	GetVersionProperty.uiMinor := 0;
	GetVersionProperty.uiServicePack := 0;
	GetVersionProperty.uiPatch := 0;
END_IF

END_FUNCTION

// Device/Application/FBs/Components/ElectricPressureBarFB
FUNCTION_BLOCK ElectricPressureBarFB IMPLEMENTS IComponentStatus
VAR_INPUT
    enable : BOOL;
END_VAR
VAR_IN_OUT

END_VAR
VAR_OUTPUT
END_VAR
VAR
    electricPressureBarMotor : FB_FestoMotor();
    delay: TON := (PT := T#1S);
    state : PRESSURE_BAR_STATES;
    enableElectricPressureBarONS : R_TRIG();
    
    _mode : DEVICE_MODES;    // Auto-SemiAuto-Manual
    _ready : BOOL;            // Ready to be controlled
    _amOpenJaw : BOOL;    // Auto Mode Open Jaw Command
    _amCloseJaw : BOOL;     // Auto Mode Close Jaw Command
END_VAR

//    Function Block: ElectricPressureBarFB
//    Description: This function block is the state machine for the electric pressure bar
//    
//    Created by: Ben Hess
//    Created Date: Monday, April 16, 2018

electricPressureBarMotor(deviceType := FML.CMMP_AS,
                                        isFPCActive := TRUE, 
                                        ptrReadFHPPRegister := ADR(%IW145), 
                                        ptrReadFPCRegister := ADR(%IW149),
                                        ptrWriteFHPPRegister := ADR(%QW82),
                                        ptrWriteFPCRegister := ADR(%QW86));                                    
electricPressureBarMotor.Execute();

delay();

//Report as ready if mode is auto and we're not faulted
_ready := (_mode = DEVICE_MODES.Auto) AND NOT (state = PRESSURE_BAR_STATES.Fault);


enableElectricPressureBarONS(CLK := enable);
IF enableElectricPressureBarONS.Q THEN
    state := PRESSURE_BAR_STATES.Idle;
END_IF

IF NOT enable THEN
        state := PRESSURE_BAR_STATES.Fault;
END_IF

CASE state OF
    PRESSURE_BAR_STATES.Idle:        IF enable AND _mode = DEVICE_MODES.SemiAuto OR (_mode = DEVICE_MODES.Auto AND _amCloseJaw) THEN
                                        state := PRESSURE_BAR_STATES.CloseJaw;
                                        _amCloseJaw := FALSE;
                                    END_IF
    
    PRESSURE_BAR_STATES.OpenJaw:    electricPressureBarMotor.ExecuteStoredProgram(1);
                                    IF electricPressureBarMotor.CommandAcknowledged THEN
                                        state := PRESSURE_BAR_STATES.OpeningJaw;
                                        Globals.electricPressureBarCount := Globals.electricPressureBarCount + 1;
                                    END_IF
        
    
    PRESSURE_BAR_STATES.OpeningJaw:    
                                    IF electricPressureBarMotor.ActiveStoredProgramNumber = 1 AND electricPressureBarMotor.InPosition THEN
                                        state := PRESSURE_BAR_STATES.JawOpened;
                                    END_IF
                                    
    PRESSURE_BAR_STATES.JawOpened:     IF _mode = DEVICE_MODES.SemiAuto THEN
                                        delay.IN := TRUE;
                                        IF delay.Q THEN
                                            state := PRESSURE_BAR_STATES.CloseJaw;
                                            delay.IN := FALSE;
                                        END_IF
                                    ELSIF _mode = DEVICE_MODES.Auto AND _amCloseJaw THEN
                                        state := PRESSURE_BAR_STATES.CloseJaw;
                                        _amCloseJaw := FALSE;
                                    END_IF
        
    PRESSURE_BAR_STATES.CloseJaw:    electricPressureBarMotor.ExecuteStoredProgram(2);
                                    IF electricPressureBarMotor.CommandAcknowledged THEN
                                        state := PRESSURE_BAR_STATES.ClosingJaw;
                                        Globals.electricPressureBarCount := Globals.electricPressureBarCount + 1;
                                    END_IF
                                    
    
    PRESSURE_BAR_STATES.ClosingJaw:    IF electricPressureBarMotor.ActiveStoredProgramNumber = 2 AND electricPressureBarMotor.InPosition THEN
                                        state := PRESSURE_BAR_STATES.JawClosed;
                                    END_IF
                                    
    PRESSURE_BAR_STATES.JawClosed:    IF _mode = DEVICE_MODES.SemiAuto THEN
                                        delay.IN := TRUE;
                                        IF delay.Q THEN
                                            state := PRESSURE_BAR_STATES.OpenJaw;
                                            delay.IN := FALSE;
                                        END_IF
                                    ELSIF _mode = DEVICE_MODES.Auto AND _amOpenJaw THEN
                                        state := PRESSURE_BAR_STATES.OpenJaw;
                                        _amOpenJaw := FALSE;
                                    END_IF
    
    PRESSURE_BAR_STATES.Fault:        ClearCommands();        
    
    
END_CASE

METHOD AutoCloseJaw
VAR_INPUT
END_VAR
_amCloseJaw := TRUE;
END_METHOD

METHOD AutoOpenJaw
VAR_INPUT
END_VAR
_amOpenJaw := TRUE;
END_METHOD

PROPERTY Mode : DEVICE_MODES
SET
_mode := Mode;
END_SET
GET
Mode := _mode;
END_GET
END_PROPERTY

PROPERTY Ready : BOOL
SET
_ready := Ready;
END_SET
GET
Ready := _ready;
END_GET
END_PROPERTY

METHOD PRIVATE ClearCommands
VAR_INPUT
END_VAR
_amCloseJaw := FALSE;
_amOpenJaw := FALSE;
END_METHOD

END_FUNCTION_BLOCK

// Device/Application/Programs/PRG_
FUNCTION_BLOCK PRG_
VAR_INPUT
END_VAR
VAR_OUTPUT
END_VAR
VAR
END_VAR

END_FUNCTION_BLOCK

// Device/Application/FBs/Components/PickAndPlaceFB
FUNCTION_BLOCK PickAndPlaceFB EXTENDS BaseComponentFB
VAR_INPUT
	XAxisMotor : IPositionableMotor;	// X Axis Motor
	YAxisMotor : IPositionableMotor;	// Y Axis Motor
	ZAxisMotor : IPositionableMotor;	// Z Axis Motor
END_VAR
VAR_OUTPUT
	state : VACUUM_PICKER_STATES;	 //State indication
END_VAR
VAR
	
	accel : INT := 2000;
	decel : INT := 2000;
	velo : INT := 2000;
	zVelo : INT := 12000;
END_VAR

//	Function Block: PickAndPlaceFB
//	Description: This provides the methods and state machine to operate the Vacuum Head pick and place machine
//	
//	Created by: Ben Hess
//	Created Date: Friday, June 1, 2018

// Run the base FB
SUPER^();

// Set up the 3 motors.

// X Axis moves out and in relative to the machine. Out is 0in, max in is 7.5in.


IF enableONS.Q THEN
    IF _mode = DEVICE_MODES.Manual THEN 
        state := VACUUM_PICKER_STATES.Manual;
    ELSE
        state := VACUUM_PICKER_STATES.Ready;
    END_IF
END_IF

IF NOT enable THEN
    state := VACUUM_PICKER_STATES.Idle;
END_IF

_ready := (_mode = DEVICE_MODES.Auto) AND NOT (state = VACUUM_PICKER_STATES.Fault);


CASE state OF
	VACUUM_PICKER_STATES.Idle :
	VACUUM_PICKER_STATES.Home :								// Move everything to home position
															XAxisMotor.MoveToPosition(6, accel,decel,velo);
															YAxisMotor.MoveToPosition(15, accel,decel,velo);
															ZAxisMotor.MoveToPosition(1, accel,decel,zVelo);
															state := VACUUM_PICKER_STATES.Homing;
															
	VACUUM_PICKER_STATES.Homing :							// Move on if all motors report ready
															IF XAxisMotor.CurrentPosition = 6
																AND YAxisMotor.CurrentPosition = 15
																AND ZAxisMotor.CurrentPosition = 1 THEN
																	state := VACUUM_PICKER_STATES.Homed;
															END_IF
															
	VACUUM_PICKER_STATES.Homed :							// 
															state :=VACUUM_PICKER_STATES.XAxisMoveIn;
															
	VACUUM_PICKER_STATES.XAxisMoveIn :						// Move XAxis in 
															XAxisMotor.MoveToPosition(0,accel,decel,velo);
															state := VACUUM_PICKER_STATES.XAxisMovingIn;
															
	VACUUM_PICKER_STATES.XAxisMovingIn :					// 
															IF XAxisMotor.CurrentPosition = 0 THEN
																state := VACUUM_PICKER_STATES.XaxisMovedIn;
															END_IF
															
	VACUUM_PICKER_STATES.XaxisMovedIn :						// 
															state := VACUUM_PICKER_STATES.VacuumTurnOn;
															
	VACUUM_PICKER_STATES.VacuumTurnOn :						// 
															state := VACUUM_PICKER_STATES.VacuumHeadDown;
															
	VACUUM_PICKER_STATES.VacuumHeadDown :					// 
															ZAxisMotor.MoveToPosition(150,accel,decel,zVelo);
															state := VACUUM_PICKER_STATES.YAxisMoveDown;
															
	VACUUM_PICKER_STATES.YAxisMoveDown :					// 
															YAxisMotor.MoveToPosition(1,accel,decel,velo);
															state := VACUUM_PICKER_STATES.VacuumHeadAndYAxisMovingDown;
															
	VACUUM_PICKER_STATES.VacuumHeadAndYAxisMovingDown :		// 
															IF YAxisMotor.CurrentPosition = 1
																AND ZAxisMotor.CurrentPosition = 150 THEN
																state := VACUUM_PICKER_STATES.VacuumHeadAndYAxisMovedDown;  
															END_IF	
															
	VACUUM_PICKER_STATES.VacuumHeadAndYAxisMovedDown :		// 
															state := VACUUM_PICKER_STATES.VacuumTurnOff;
															
	VACUUM_PICKER_STATES.VacuumTurnOff :					// 
															state := VACUUM_PICKER_STATES.ConveyorTurnOn;
															
	VACUUM_PICKER_STATES.ConveyorTurnOn :					// 
															state := VACUUM_PICKER_STATES.ConveyorMoving;
															
	VACUUM_PICKER_STATES.ConveyorMoving :					// 
															state := VACUUM_PICKER_STATES.ConveyorDone;
															
	VACUUM_PICKER_STATES.ConveyorDone :						// 
															state := VACUUM_PICKER_STATES.Ready;
															
	VACUUM_PICKER_STATES.Fault :							// 
																													
	
	VACUUM_PICKER_STATES.Ready :							IF semiAutoModeSelected THEN
																state := VACUUM_PICKER_STATES.Home;
															END_IF
	VACUUM_PICKER_STATES.Manual :
END_CASE

END_FUNCTION_BLOCK

// Device/Application/ObjectHandling/IExhaustable
INTERFACE IExhaustable EXTENDS IAllObjects

END_INTERFACE

// Library Information/GetLibVersion
// This function has been automatically generated from the project information.
FUNCTION GetLibVersion : VERSION
VAR_INPUT
	
END_VAR

GetLibVersion.uiMajor := 0;
GetLibVersion.uiMinor := 9;
GetLibVersion.uiServicePack := 13;
GetLibVersion.uiPatch := 2;

END_FUNCTION

// Device/Application/FBs/Fault/FB_InternalLogger
FUNCTION_BLOCK FB_InternalLogger IMPLEMENTS IMachineLogger
VAR_INPUT
END_VAR
VAR_OUTPUT
END_VAR
VAR
	//loggedItems : ARRAY[0..500] OF FaultLogType;
	loggedItems : ARRAY[0..GLobals.MAX_LOGGED_ITEMS] OF LogMessageType;
	numOfLogEntries : UINT;
	logFull : BOOL;
	RTC : FB_GetTime();
	clearLog : BOOL;
	i : UINT;
END_VAR

//	Function Block: FB_Logger
//	Description: This is an internal logger for reference within Codesys.  It is an array that can be displayed on the TargetVisu/WebVisu 
//	
//	Created by: Ben Hess
//	Created Date: Tuesday, September 11, 2018

RTC();

IF clearLog THEN
	FOR i := 0 TO numOfLogEntries BY 1 DO
		loggedItems[i].logMessage := '';
		loggedItems[i].logTime := DT#1970-1-1-1:0:0;
	END_FOR
	numOfLogEntries := 0;
	logFull := FALSE;
	clearLog := FALSE;
END_IF

PROPERTY InstanceName : STRING
GET
END_GET
END_PROPERTY

METHOD AddLogItem
VAR_INPUT
	message : STRING;
END_VAR
FOR i := Globals.MAX_LOGGED_ITEMS -1 TO 1 BY -1 DO
		loggedItems[i] := loggedItems[i-1];
END_FOR

loggedItems[0].logMessage := message;
loggedItems[0].logTime := RTC.currentDateAndTime;
END_METHOD

END_FUNCTION_BLOCK

// Project Information/GetNumberProperty
// This function has been automatically generated from the project information.
{attribute 'signature_flag' := '1073741824'}
{attribute 'register_in_runtime'}
FUNCTION GetNumberProperty : DINT
VAR_INPUT
	stKey: WSTRING;
END_VAR

GetNumberProperty := 0;

END_FUNCTION

// Library Information/GetLibVersionNumber
// This function has been automatically generated from the project information.
FUNCTION GetLibVersionNumber : DWORD
VAR_INPUT
	
END_VAR

GetLibVersionNumber := 593154;

END_FUNCTION

// Device/Application/FBs/Motors/Applied Motion/Modbus Commands/FB_SendOpcodeCommandAppliedMotionRTU
FUNCTION_BLOCK FB_SendOpcodeCommandAppliedMotionRTU
VAR_INPUT
    Parameter1 : WORD := 0;        //QX Parameter 1
    Parameter2 : WORD := 0;        //QX Parameter 2
    Parameter3 : WORD := 0;        //QX Parameter 3
    Parameter4 : WORD := 0;        //QX Parameter 3
    Parameter5 : WORD := 0;        //QX Parameter 3
    opcode : STEP_SERVO_OPCODES;    //Opcode to perform
END_VAR
VAR_IN_OUT
    opcodeWithArgumentsSettingsBuffer : ARRAY[0..1] OF WORD;
END_VAR

VAR_OUTPUT
    xDone : BOOL;        //Successfully performed action
    triggerOpcodeWrite : BOOL;
END_VAR
VAR
    QXCommandState : OPCODE_MODBUS_COMMAND_STATES;
    sendBuffer : ARRAY [0 .. 5] OF WORD;            //Array of registers to send
    xExecute : BOOL;
    xExecuteONS : R_TRIG();
END_VAR


xExecuteONS(CLK := xExecute);
IF xExecuteONS.Q THEN
    xDone := FALSE;
END_IF    
                                
CASE QXCommandState OF
    OPCODE_MODBUS_COMMAND_STATES.Idle :                    //Move on to Send Parameters
                                                        IF xExecute THEN
                                                            QXCommandState := OPCODE_MODBUS_COMMAND_STATES.SendOpcodeAndParameters;
                                                        END_IF
                                                        xExecute := FALSE;
                                
    OPCODE_MODBUS_COMMAND_STATES.SendOpcodeAndParameters :            
                                                        //Setup parameter registers to send to drive
                                                        triggerOpcodeWrite := TRUE;
                                                        QXCommandState := OPCODE_MODBUS_COMMAND_STATES.WaitAfterOpcodeAndParametersSent;
                                                        
                                                        
    OPCODE_MODBUS_COMMAND_STATES.WaitAfterOpcodeAndParametersSent :
                                                        //Wait for confimation
                                                            xDone := TRUE;
                                                            triggerOpcodeWrite := FALSE;
                                                            QXCommandState := OPCODE_MODBUS_COMMAND_STATES.Idle;
                                                
    OPCODE_MODBUS_COMMAND_STATES.Fault :                    
                                                        //Move on to Send Parameters
                                                        IF xExecute THEN
                                                            QXCommandState := OPCODE_MODBUS_COMMAND_STATES.SendOpcodeAndParameters;
                                                        END_IF
                                                        xExecute := FALSE;
END_CASE

METHOD Execute
VAR_INPUT
END_VAR
xExecute := TRUE;
END_METHOD

END_FUNCTION_BLOCK

// Device/Application/FBs/SerialMotorTestFB
FUNCTION_BLOCK SerialMotorTestFB
VAR_INPUT
    runMotorPB : BOOL;
END_VAR
VAR_OUTPUT
END_VAR
VAR
    //testMotor : FB_AppliedMotionStepServoRTU();    
    //orientalMotor : FB_OrientalAZDrive();
END_VAR

(*
orientalMotor(modbusInBuffer := OrientalMotorModbusRead,
                stepsPerInchSetpoint := 2122,
                reversePolarity := FALSE,
                operatingCurrentDefault := 100,
                modbusCommandOutBuffer := OrientalMotorCommandWrites,
                modbusParametersOutBuffer := OrientalMotorParameterWrites,
                triggerCommandWrite => OrientalMotorTriggerCommandWrite,
                triggerParameterWrite => OrientalMotorTriggerParameterWrite);                
orientalMotor.Execute();
*)


IF runMotorPB THEN
    //testMotor.MoveDistance(12,100,100,215);
    //testMotor.HomeNow();
    
    //orientalMotor.MoveDistance(12,10000,10000,10000);
    runMotorPB := FALSE;
END_IF

END_FUNCTION_BLOCK

// Device/Application/Event Handlers/PrepareOnlineChange
FUNCTION PrepareOnlineChange : DWORD
VAR_IN_OUT
	EventPrm: CmpApp.EVTPARAM_CmpApp;
END_VAR
VAR
END_VAR

SaveValues();

END_FUNCTION

// Device/Application/Event Handlers/PrepareStop
FUNCTION PrepareStop : DWORD
VAR_IN_OUT
	EventPrm: CmpApp.EVTPARAM_CmpAppStop;
END_VAR
VAR
END_VAR

SaveValues();

END_FUNCTION

// Device/Application/ObjectHandling/IFault_1
INTERFACE IFault_1 EXTENDS IAllObjects

METHOD Ack
VAR_INPUT
END_VAR
END_METHOD

METHOD Trigger
VAR_INPUT
END_VAR
END_METHOD

END_INTERFACE

// Device/Application/ObjectHandling/FB_CollectionHandlerFaults
FUNCTION_BLOCK FB_CollectionHandlerFaults
VAR_INPUT
END_VAR
VAR
	Collection: ARRAY[0..GlobalObjects.MAX_FAULTS] OF IFault; // object array
	ObjNames   : ARRAY[0..GlobalObjects.MAX_FAULTS] OF STRING;
	_ArrayOver   : BOOL;
	_BadObj      : INT;
	_DupeObj   : INT;
	_OverObj   : INT;
	_TotalObj   : UINT;
END_VAR

METHOD AckAll
VAR_INPUT
END_VAR
VAR
	J : UINT;
END_VAR
FOR J:= 0 TO _TotalObj - 1 DO
	Collection[J].Ack();
END_FOR
END_METHOD

METHOD AddObject
VAR_INPUT
	Obj   : IFault;
END_VAR
VAR
	J   : UINT;
END_VAR
FOR J:= 0 TO _TotalObj DO
	IF Collection[J] = Obj THEN
		// object pointer matches - dupe!
		_DupeObj:= _DupeObj + 1;
		RETURN;
	END_IF
END_FOR
   
IF _TotalObj < GlobalObjects.MAX_FAULTS THEN
	Collection[_TotalObj]:= Obj;
	ObjNames[_TotalObj]:= Obj.InstanceName;
	_TotalObj:= _TotalObj + 1;
ELSE
	_ArrayOver:= TRUE;
	_OverObj:= _OverObj + 1;
END_IF
END_METHOD

END_FUNCTION_BLOCK

// Device/Application/FBs/Components/HeadRaiseLowerFB
FUNCTION_BLOCK HeadRaiseLowerFB
VAR_INPUT
	upperLimitProx : BOOL;
	lowerLimitProx : BOOL;
	raiseCommand : BOOL;
	lowerCommand : BOOL;
END_VAR
VAR_OUTPUT
	raiseOutput : BOOL;
	lowerOutput : BOOL;
END_VAR
VAR
END_VAR

IF raiseCommand AND NOT upperLimitProx THEN
	raiseOutput := TRUE;
ELSE
	raiseOutput := FALSE;
END_IF

IF lowerCommand AND NOT lowerLimitProx THEN
	lowerOutput := TRUE;
ELSE
	lowerOutput := FALSE;
END_IF

END_FUNCTION_BLOCK

// Device/Application/ObjectHandling/FB_CollectionHandlerExecutable
FUNCTION_BLOCK FB_CollectionHandlerExecutable
VAR_INPUT
END_VAR
VAR
	Collection: ARRAY[0..GlobalObjects.MAX_EXECUTEABLE] OF IExecuteAutomatically; // object array
	ObjNames   : ARRAY[0..GlobalObjects.MAX_EXECUTEABLE] OF STRING;
	_ArrayOver   : BOOL;
	_BadObj      : INT;
	_DupeObj   : INT;
	_OverObj   : INT;
	_TotalObj   : UINT;
END_VAR

//	Function Block: FB_CollectionHandlerExecutable
//	Description: This collection handler stores executable FB's to an array 
//				 and has a method to execute them all on demand
//	Created by: Ben Hess
//	Created Date: Friday, September 7, 2018

METHOD ExecuteAll
VAR_INPUT
END_VAR
VAR
	Cast : IExecuteAutomatically;
	J : UINT;
END_VAR
// For each executable objest in the array, run its "Execute()" method
FOR J:= 0 TO _TotalObj - 1 DO
	IF (__QUERYINTERFACE(Collection[J], Cast)) THEN
		Cast.Execute();
	ELSE 
		RETURN;
	END_IF
END_FOR
END_METHOD

METHOD AddObject
VAR_INPUT
	Obj   : IExecuteAutomatically;
END_VAR
VAR
	I   : UINT;
	J : UINT;
END_VAR
// Add the active fault to the array 
FOR J:= 0 TO _TotalObj DO
	IF Collection[J] = Obj THEN
		// object pointer matches - it's already in here
		RETURN;
	END_IF
END_FOR
   
IF _TotalObj < GlobalObjects.MAX_EXECUTEABLE THEN
	Collection[_TotalObj]:= Obj;
	ObjNames[_TotalObj]:= Obj.InstanceName;
	_TotalObj:= _TotalObj + 1;
ELSE
	_ArrayOver:= TRUE;
	_OverObj:= _OverObj + 1;
END_IF
END_METHOD

END_FUNCTION_BLOCK

// Device/Application/Interfaces/ISupervisor
INTERFACE ISupervisor

METHOD NotifyMachineFaulted
VAR_INPUT
END_VAR
END_METHOD

METHOD MakeReady
VAR_INPUT
END_VAR
END_METHOD

END_INTERFACE

(* text list System (id | default)
  Apr | Apr
  April | April
  Aug | Aug
  August | August
  Dec | Dec
  December | December
  Feb | Feb
  February | February
  Fri | Fri
  Friday | Friday
  Jan | Jan
  January | January
  Jul | Jul
  July | July
  Jun | Jun
  June | June
  Mar | Mar
  March | March
  May | May
  May_3Letter | May
  Mon | Mon
  Monday | Monday
  Nov | Nov
  November | November
  Oct | Oct
  October | October
  Sat | Sat
  Saturday | Saturday
  Sep | Sep
  September | September
  Sun | Sun
  Sunday | Sunday
  Thu | Thu
  Thursday | Thursday
  Tue | Tue
  Tuesday | Tuesday
  Wed | Wed
  Wednesday | Wednesday
   |  *)
